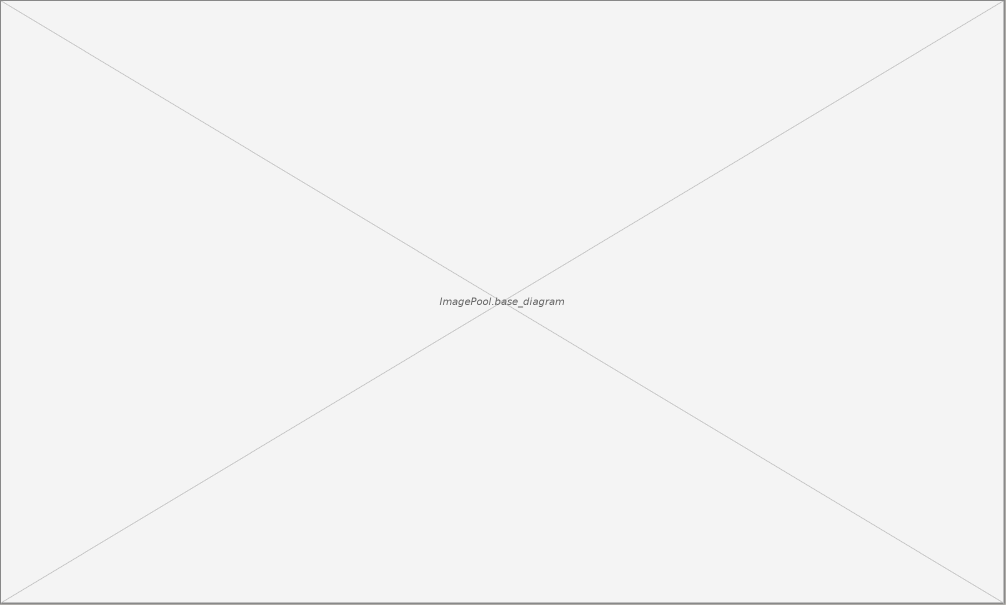
VISUALIZATION TESimMain  // 1006x605
    Image (0,0 1004x603), image: ImagePool.base_diagram
END_VISUALIZATION

(* stored: Version 1.1.0.1, ProductVersion 3.1.0.36
   Visu TESimMain: Id {50d0fa6c-6a14-4701-b805-7bcabed7b14e} *)
